PROGRAM FB_IKR270
VAR
	AO:INT;
	rPRESS:REAL;
	xPRESS_OK:BOOL;
	xHV_DIS:BOOL;
END_VAR

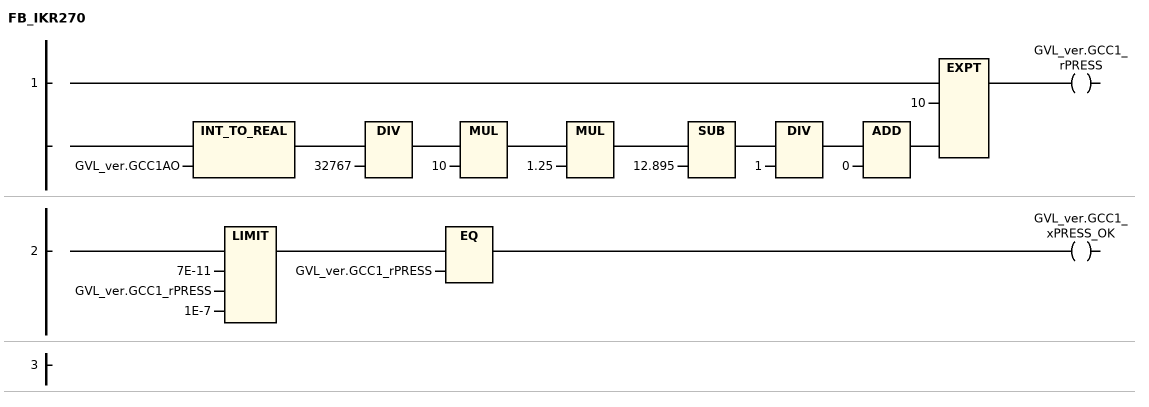
// NETWORK 1
GVL_ver.GCC1_rPRESS := EXPT(10, (((INT_TO_REAL(GVL_ver.GCC1AO) / 32767) * 10) * 1.25 - 12.895) / 1 + 0);

// NETWORK 2
GVL_ver.GCC1_xPRESS_OK := LIMIT(7E-11, GVL_ver.GCC1_rPRESS, 1E-7) = GVL_ver.GCC1_rPRESS;

// NETWORK 3

END_PROGRAM

(* stored: Version 1.1.0.1, ProductVersion 3.1.4022.3
   POU FB_IKR270: Id {51b9548d-8cab-45b0-b18e-b66fb74df604}, SpecialFunc None *)
